// TIA Portal V15.1 export
// export: Created 2026-01-15T16:29:35.7148256Z, ExportSetting WithDefaults, WithReadOnly, DisplayName Totally Integrated Automation Portal, DisplayVersion V15.1 Update 8, DisplayName TIA Portal Openness, DisplayVersion V15.1 Update 8, DisplayName STEP 7 Professional, DisplayVersion V15.1 Update 8, DisplayName WinCC Advanced, DisplayVersion V15.1 Update 8
ORGANIZATION_BLOCK "Main"   // OB123, LAD, ProgramCycle
TITLE = "Main Program Sweep (Cycle)"
{ S7_Optimized_Access := 'TRUE' }
VERSION : 0.1
// stored: AutoNumber true, CodeModifiedDate 2026-01-15T16:25:55.6274482Z, CompileDate 2026-01-15T16:25:55.6406611Z, ConstantName OB_Main, CreationDate 2026-01-15T16:14:49.4586784Z, EventClass Program cycle, HandleErrorsWithinBlock false, InterfaceModifiedDate 2026-01-15T16:25:47.5430699Z, IsConsistent true, IsIECCheckEnabled false, IsKnowHowProtected false, IsWriteProtected false, ModifiedDate 2026-01-15T16:25:55.6274482Z, ParameterModified 2008-07-21T16:55:08.419547Z, PLCSimAdvancedSupport false, PriorityNumber 1, ProcessImagePartNumber 65535, SetENOAutomatically False, StructureModified 2008-07-21T16:55:08.419547Z
   VAR_INPUT
      Initial_Call : Bool;   // Initial call of this OB
      Remanence : Bool;   // =True, if remanent data are available
   END_VAR
BEGIN
END_ORGANIZATION_BLOCK
